PROGRAM MAIN
VAR
	StateMachine: FB_StateMachine;
	Visualization: FB_Visualization;
END_VAR

StateMachine(bStart:= GVL.bStart, bStop:= GVL.bStop, bLimitLeft:= GVL.bLimitLeft, bLimitRight:= GVL.bLimitRight );
Visualization(bMovingRight:= StateMachine.bMovingRight, bMovingLeft:=StateMachine.bMovingLeft);
GVL.bLimitLeft := Visualization.bLimitLeft;
GVL.bLimitRight := Visualization.bLimitRight;

END_PROGRAM

(* stored: Version 1.1.0.1, ProductVersion 3.1.4024.12
   POU MAIN: Id {add9e90c-83f4-422c-9a2b-4e12fd816484}, SpecialFunc None *)
